FUNCTION_BLOCK animacaoEquipamento (* Basic Function Block Type *)
  (* Standard: 61499-2 *)
  (* Version 0.0, 14/01/2026, Schneider Electric, Template *)
  PACKAGE Hidryco.HidrycoLib;
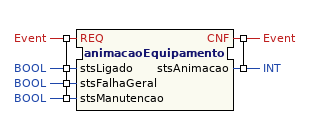
  EVENT_INPUT
    REQ WITH stsFalhaGeral, stsManutencao, stsLigado; (* Normal Execution Request *)
  END_EVENT
  EVENT_OUTPUT
    CNF WITH stsAnimacao; (* Execution Confirmation *)
  END_EVENT
  VAR_INPUT
    stsLigado : BOOL; (* Input event qualifier *)
    stsFalhaGeral : BOOL;
    stsManutencao : BOOL;
  END_VAR
  VAR_OUTPUT
    stsAnimacao : INT; (* Output event qualifier *)
  END_VAR
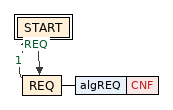
  EC_STATES
    START; (* Initial State *)
    REQ : algREQ -> CNF;
  END_STATES
  EC_TRANSITIONS
    START TO REQ := REQ;
    REQ TO START := 1;
  END_TRANSITIONS
  ALGORITHM algREQ IN ST:
IF stsManutencao THEN
    stsAnimacao := 3;
ELSIF stsFalhaGeral THEN
    stsAnimacao := 2;
ELSIF stsLigado THEN
    stsAnimacao := 1;
ELSE
    stsAnimacao := 0;
END_IF;
;
  END_ALGORITHM
END_FUNCTION_BLOCK
